// TIA Portal V17 export
// export: Created 2024-09-02T12:50:24.7249525Z, ExportSetting WithDefaults, DisplayName Totally Integrated Automation Portal, DisplayVersion V17, DisplayName TIA Portal Openness, DisplayVersion V17, DisplayName TIA Portal Version Control Interface, DisplayVersion V17, DisplayName STEP 7 Professional, DisplayVersion V17, DisplayName STEP 7 Safety, DisplayVersion V17, DisplayName WinCC Professional, DisplayVersion V17
DATA_BLOCK "Energy_Counter"   // DB2000
{ S7_Optimized_Access := 'TRUE' }
VERSION : 0.1
// stored: AutoNumber false, DBAccessibleFromOPCUA true, IsOnlyStoredInLoadMemory false, IsRetainMemResEnabled false, IsWriteProtectedInAS false, MemoryReserve 100
   VAR
      Bufor_Energy_Shift : LReal;
      Bufor_Energy_Day : LReal;
      Bufor_Energy_Week : LReal;
      Bufor_Energy_Month : LReal;
      Bufor_Energy_Year : LReal;
      Bufor_Air_Shift : LReal;
      Bufor_Air_Day : LReal;
      Bufor_Air_Week : LReal;
      Bufor_Air_Month : LReal;
      Bufor_Air_Year : LReal;
      Reset_Total : Bool;
      Reset_Time_stamp : Bool;
      Total_Part : Int;
      Last_Mounth_Part : Int;
      Bufor_Last_Mounth_Part : Int;
      Counter_Part_Total : IEC_COUNTER;
      Counter_Part_Last_Mounth : IEC_COUNTER;
      Trigger_Neg : Array[0..19] of Bool;
      Trigger_Pos : Array[0..19] of Bool;
      REAL_TIME_DATE : DTL;
      Energy_Out_Structure : Struct
         Total : LReal;
         Shift : LReal;
         Day : LReal;
         Week : LReal;
         Last_Week : LReal;
         Month : LReal;
         Last_Month : LReal;
         Year : LReal;
         per_Part : LReal;
      END_STRUCT;
      Air_Out_Structure : Struct
         Total : LReal;
         Shift : LReal;
         Day : LReal;
         Week : LReal;
         Last_Week : LReal;
         Month : LReal;
         Last_Month : LReal;
         Year : LReal;
         per_Part : LReal;
      END_STRUCT;
      TON : Struct
         Restart_Period : IEC_TIMER;
         Restart_Total : IEC_TIMER;
      END_STRUCT;
      Last_Total_Restart : DTL;
      Last_Period_Restart : DTL;
   END_VAR
BEGIN
END_DATA_BLOCK
